// TIA Portal V16 export
// export: Created 2022-02-04T14:40:19.7253243Z, ExportSetting WithDefaults, DisplayName Totally Integrated Automation Portal, DisplayVersion V16 Update 1, DisplayName TIA Portal Version Control Interface, DisplayVersion V16, DisplayName TIA Portal Openness, DisplayVersion V16, DisplayName SINAMICS Startdrive Advanced, DisplayVersion V16 Update 5, DisplayName SINAMICS Startdrive G130, G150, S120, S150, SINAMICS MV, S210, DisplayVersion V16 Update 5, DisplayName SINAMICS Startdrive G110M, G120, G120C, G120D, G120P, G115D, DisplayVersion V16 Update 5, DisplayName STEP 7 Professional, DisplayVersion V16, DisplayName STEP 7 Safety, DisplayVersion V16, DisplayName WinCC Advanced, DisplayVersion V16, DisplayName SIMATIC Visualization Architect, DisplayVersion V16
DATA_BLOCK "VELOCITY"   // DB19
VERSION : 0.1
// stored: AutoNumber true, IsOnlyStoredInLoadMemory false, IsWriteProtectedInAS false
   VAR RETAIN
      GeneralSpeed : Real;   // Общая скорость линии
      koef_M_332 : Real := 0.4;   // сброс с рольганга
      koef_M_333 : Real := 0.24;   // рольганг брака
      koef_M_334 : Real := 0.2;   // набор слоя
      koef_M_335 : Real := 0.12;   // вилы
      koef_M_336 : Real := 0.2;   // лифт
      koef_M_212 : Real := 0.2;   // лифт загрузки
      koef_M_213 : Real := 0.45;   // наклонный транспортер
      koef_M_222 : Real := 0.09;   // главная горка
      koef_M_231 : Real := 0.12;   // Ролики прибортовщики
      koef_M_325 : Real := 0.7;   // Довод слоя
      koef_M_225 : Real := 0.142;   // Транспортер с бобышками
      koef_M_223 : Real := 0.3;   // зона оценки
      koef_M_232 : Real := 0.25;   // лифт ПФМ
   END_VAR
BEGIN
END_DATA_BLOCK
